// TIA Portal V17 export
// export: Created 2024-09-15T12:30:13.8156718Z, ExportSetting WithDefaults, DisplayName Totally Integrated Automation Portal, DisplayVersion V17, DisplayName TIA Portal Openness, DisplayVersion V17, DisplayName TIA Portal Version Control Interface, DisplayVersion V17, DisplayName STEP 7 Professional, DisplayVersion V17, DisplayName STEP 7 Safety, DisplayVersion V17, DisplayName WinCC Professional, DisplayVersion V17
DATA_BLOCK "Simulation_Variables"   // DB45
{ S7_Optimized_Access := 'FALSE' }
VERSION : 0.1
// stored: AutoNumber true, DBAccessibleFromOPCUA true, DBAccessibleFromWebserver true, IsOnlyStoredInLoadMemory false, IsWriteProtectedInAS false
   VAR
      HBW_Horizontal_Encoder : Int;
      HBW_Vertical_Encoder : Int;
      HBW_Gripper_Pos_In : Bool;
      HBW_Gripper_Pos_Out : Bool;
      HBW_Gripper_Forward : Bool;
      HBW_Gripper_Backward : Bool;
      HBW_Gripper_PWM : Int;
      HBW_Belt_Pos_In : Bool;
      HBW_Belt_Pos_Out : Bool;
      HBW_Belt_Forward : Bool;
      HBW_Belt_Backward : Bool;
      HBW_Belt_PWM : Int;
      HBW_Product_1_Color : Byte;
      HBW_Product_2_Color : Byte;
      HBW_Product_3_Color : Byte;
      HBW_Product_4_Color : Byte;
      HBW_Product_5_Color : Byte;
      HBW_Product_6_Color : Byte;
      HBW_Product_7_Color : Byte;
      HBW_Product_8_Color : Byte;
      HBW_Product_9_Color : Byte;
      HBW_Product_Bind : Byte;
      HBW_Product_InOut_Color : Byte;
      HBW_Product_InOut_Toggle : Bool;
      VGR_Rotate_Encoder : Int;
      VGR_Vertical_Encoder : Int;
      VGR_Horizontal_Encoder : Int;
      VGR_Product_Color : Byte;
   END_VAR
BEGIN
END_DATA_BLOCK
